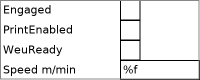
VISUALIZATION _VISU_PrintModule_main  // 200x80
VAR_IN_OUT
  mInst : FB_PrintModule;
END_VAR
    RoundedRectangle (120,0 20x20), colour toggle: PRG_PRINT.bL_Engaged[mInst._nIdx]
    Rectangle (0,0 120x20), "Engaged"
    Rectangle (0,20 120x20), "PrintEnabled"
    RoundedRectangle (120,20 20x20), colour toggle: PRG_PRINT.bL_PmPrintEnabled[mInst._nIdx]
    Rectangle (0,60 120x20), "Speed m/min"
    Rectangle (120,60 80x20), "%f", text variable: PRG_PRINT.fL_SpeedInMpMin[mInst._nIdx]
    RoundedRectangle (120,40 20x20), colour toggle: PRG_MACHINE.bO_WEUReady[mInst._nIdx]
    Rectangle (0,40 120x20), "WeuReady"
END_VISUALIZATION

(* stored: Version 1.1.0.1, ProductVersion 3.1.4024.9
   Visu _VISU_PrintModule_main: Id {1c33c1d3-4cba-4983-923f-6027f0964b30} *)
